// TIA Portal V18 export
VAR_GLOBAL   // PLC tag table "Selector"
   Anti_Phase AT %I0.0 : Bool;
   Reset AT %I0.1 : Bool;
   Emergency_Stop AT %I0.2 : Bool;
   Auto_Manual AT %Q0.0 : Bool;
   Command_Auto AT %Q0.1 : Bool;
   Command_Manual AT %Q0.2 : Bool;
END_VAR
